DEVICE_TYPE {name} (* Device '{name}' *)
  (* Standard: 61499-2 *)
  (* Version 0.1, {date}, {author}, NetAllied, Initial creation. *)
END_DEVICE_TYPE
